{attribute 'GeneratedUsingTerminal: EPP5101-0002-0016'}
{attribute addProperty BoxType "EPP5101-0002-0016"}
{attribute addProperty Id "StatusAT %I*Status_3A9E406C12Counter_valueAT %I*UINT2Latch_valueAT %I*UINT2"}
{attribute addProperty CRC "4109931907"}
{attribute addProperty Size "16"}
TYPE ENC_Status_compact_F4F89583 EXTENDS InputBase_8311D824 :
STRUCT
	{attribute addProperty Name "Status"}
	Status AT %I* : Status_3A9E406C;
	{attribute addProperty Name "Counter_value"}
	Counter_value AT %I* : UINT;
	{attribute addProperty Name "Latch_value"}
	Latch_value AT %I* : UINT;
END_STRUCT
END_TYPE

(* stored: Version 1.2.0.0, ProductVersion 3.1.4024.11
   DUT ENC_Status_compact_F4F89583: Id {1ce3f2e9-faaa-4f54-b1a1-ea11c1613037} *)
